INTERFACE ISumCollector

METHOD addValue
VAR_INPUT
END_VAR
END_METHOD

PROPERTY sum : LINT
GET
END_GET
SET
END_SET
END_PROPERTY

END_INTERFACE

(* stored: Version 1.1.0.1
   Itf ISumCollector: Id {9423d3f1-8ee5-419c-8020-86e79515db95}
   Method addValue: Id {7b44a895-3cdf-4088-a928-8786d14bbdbf}
   Property sum: Id {0ed31d92-c052-4d73-971e-507d8cf647ce}
   Get Get: Id {5e68f898-8ecd-463b-9996-2c7b4db4f021}
   Set Set: Id {3d1ce1e6-d6a9-4459-aae3-337db5d6fd38} *)
